(* Logix 5000 project; controller ARS14002_PLC vendor 1 type 14 code 218 rev 30.11; software revision 30.01; part 4 of 13 *)
(* tags used below, declared in another part *)
   ARGON_FROM_TK1100A : BOOL;
   ARGON_FROM_TK700 : BOOL;
   ARS14002_PLC_LEDStatus : INT;
   ARS14002_PLC_Slot1Status : INT;
   ARS14002_PLC_Slot2Status : INT;
   ARS14002_PLC_Slot3Status : INT;
   ARS14002_PLC_Slot4Status : INT;
   ARS14002_PLC_Slot5Status : INT;
   ARS14002_PLC_Status : INT;
   ARS_AUTORETURN_IGNORE_AUTO : BOOL;   // Turns furnace return autoswitch on or off
   ARS_COLLECT : BOOL;
   ARS_COLLECT_AUTO : BOOL;
   ARS_IDLE : BOOL;   // **future use
   ARS_Manual_Backfill : BOOL;   // **future use
   ARS_READY_TO_RECEIVE : BOOL;
   ARS_READY_TO_SEND : BOOL;
   ARS_RETURN : BOOL;
   ARS_RETURN_AUTO : BOOL;
   ARS_STANDBY : BOOL;
   AT2_ATOMIZE_FLOW : REAL;
   AT2_ATOMIZE_FLOW_ATOMIZE_SP : REAL;
   AT2_AtomizingStatus_OSF_OB : BOOL;
   AT2_AtomizingStatus_OSF_SB : BOOL;
   AT2_AtomizingStatus_OSR_OB : BOOL;
   AT2_AtomizingStatus_OSR_SB : BOOL;
   AT2_CHAMBER_PRESSURE : REAL;
   AT2_CHAMBER_PRESSURE_SP : REAL;
   AT2_COMM_STATUS_CONS : BOOL;
   AT2_COMM_STATUS_PROD : BOOL;
   AT2_END_ATOMIZATION : BOOL;
   AT2_HIBON_RUNNING : BOOL;
   AT2_INLET_FLOW : REAL;
   AT2_INLET_FLOW_BACKFILL_SP : REAL;
   AT2_INLET_VALVE_OPEN : BOOL;
   AT2_PLANT_ATOMIZING : BOOL;
   AT2_PLANT_BACKFILL : BOOL;
   AT2_PLANT_BACKFILL_TIMEOUT_TMR : TIMER;
   AT2_PLANT_COLLECT_AUTO : BOOL;
   AT2_PLANT_COMMLOSS : BOOL;
   AT2_PLANT_POST_ATOMIZE_TON : TIMER;
   AT2_PLANT_POST_ATOMIZING : BOOL;
   AT2_PLANT_POST_ATOMIZING_CHAMBER_SP : REAL;
   AT2_PLANT_RETURN_AUTO : BOOL;
   AT2_PRAXAIR_PRESSURE : REAL;
   AT2_PRAXAIR_PRESSURE_RETURN_SPH : REAL;
   AT2_PRAXAIR_PRESSURE_RETURN_SPL : REAL;
   AT2_START_ATOMIZATION : BOOL;
   AT2_V1_OPEN : BOOL;
   AT3_ATOMIZE_FLOW : REAL;
   AT3_ATOMIZE_FLOW_ATOMIZE_SP : REAL;
   AT3_ATOMIZE_VALVE_OPEN : BOOL;
   AT3_AtomizingStatus_OSF_OB : BOOL;
   AT3_AtomizingStatus_OSF_SB : BOOL;
   AT3_AtomizingStatus_OSR_OB : BOOL;
   AT3_AtomizingStatus_OSR_SB : BOOL;
   AT3_CHAMBER_PRESSURE : REAL;
   AT3_CHAMBER_PRESSURE_SP : REAL;
   AT3_COMM_STATUS_CONS : BOOL;
   AT3_COMM_STATUS_PROD : BOOL;
   AT3_END_ATOMIZATION : BOOL;
   AT3_HIBON_RUNNING : BOOL;
   AT3_INLET_FLOW : REAL;
   AT3_INLET_FLOW_BACKFILL_SP : REAL;
   AT3_INLET_VALVE_OPEN : BOOL;
   AT3_PLANT_ATOMIZING : BOOL;
   AT3_PLANT_BACKFILL : BOOL;
   AT3_PLANT_BACKFILL_TIMEOUT_TMR : TIMER;
   AT3_PLANT_COLLECT_AUTO : BOOL;
   AT3_PLANT_COMMLOSS : BOOL;
   AT3_PLANT_POST_ATOMIZE_TON : TIMER;
   AT3_PLANT_POST_ATOMIZING : BOOL;
   AT3_PLANT_POST_ATOMIZING_CHAMBER_SP : REAL;
   AT3_PLANT_RETURN_AUTO : BOOL;
   AT3_V1_OPEN : BOOL;
   Cold_Box_Idle : BOOL;   // **future use
   CP_PumpUp : BOOL;
   CP_PumpUp_PressurePermissive : BOOL;
   CYCLE_TIME_AT2_MIN : DINT;
   CYCLE_TIME_AT3_MIN : DINT;
   CYCLE_TIME_PILOT_MIN : DINT;
   CYCLE_TIME_REM_AT2_MIN : REAL;
   CYCLE_TIME_REM_AT3_MIN : REAL;
   CYCLE_TIME_REM_PILOT_MIN : REAL;
   ESTOP_1 : BOOL;   // Pump Skid E-Stops
   ESTOP_2 : BOOL;   // FAN/HXR E-Stops
   ESTOP_HMI : BOOL;
   ESTOP_PL : CM_DO_GENERIC;
   ESTOP_ResetReq : BOOL;
   ESTOP_TRIP : BOOL;
   EW_TEST_ATOMIZE : BOOL;
   FCV_1001 : CM_AO_VLV;
   FCV_1002 : CM_AO_VLV;
   FCV_202 : CM_AO_VLV;
   FT_904 : CM_AI_SCL;
   FVNR550_CommFlt_TON : TIMER;
   FVNR550_COMMLOSS : BOOL;
   FVNR550_L1Current_HoldingRegister : DINT;
   FVR800C_CommFlt_TON : TIMER;
   FVR800C_COMMLOSS : BOOL;
   FVR800C_L1Current_HoldingRegister : DINT;
   FVR800D_CommFlt_TON : TIMER;
   FVR800D_COMMLOSS : BOOL;
   FVR800D_L1Current_HoldingRegister : DINT;
   FVR_800C_COMMLOSS : BOOL;
   FVR_800C_EN : BOOL;
   FVR_800C_ManStartReq : BOOL;
   FVR_800C_ST : BOOL;
   FVR_800D_COMMLOSS : BOOL;
   FVR_800D_EN : BOOL;
   FVR_800D_ManStartReq : BOOL;
   FVR_800D_ST : BOOL;
   HEAT_TIMER1 : TIMER;
   HEAT_TIMER1_MIN : DINT;
   HEAT_TIMER1_MS : DINT;
   HEAT_TIMER1_SEC : DINT;
   HEAT_TIMER_AT2 : TIMER;
   HEAT_TIMER_AT2_MIN : DINT;
   HEAT_TIMER_AT2_MS : DINT;
   HEAT_TIMER_AT2_SEC : DINT;
   HEAT_TIMER_AT3 : TIMER;
   HEAT_TIMER_AT3_MIN : DINT;
   HEAT_TIMER_AT3_MS : DINT;
   HEAT_TIMER_AT3_SEC : DINT;
   HEAT_TIMER_PILOT : TIMER;
   HEAT_TIMER_PILOT_MIN : DINT;
   HEAT_TIMER_PILOT_MS : DINT;
   HEAT_TIMER_PILOT_SEC : DINT;
   MANUAL_ARS_LOCKOUT : BOOL;
   MCP_SLOT1_ERROR : BOOL;
   MCP_SLOT2_ERROR : BOOL;
   MCP_SLOT3_ERROR : BOOL;
   MCP_SLOT4_ERROR : BOOL;
   MCP_SLOT5_ERROR : BOOL;
   MODE_ATOMIZE : BOOL;
   MODE_IDLE : BOOL;
   MODE_STANDBY_IDLE : BOOL;
   MODE_STANDBY_PUMPUP : BOOL;
   OFF_TIMER_AT2 : TIMER;
   OFF_TIMER_AT3 : TIMER;
   OFF_TIMER_PILOT : TIMER;
   P_800C_Fault : BOOL;
   P_800D_Fault : BOOL;
   PDT_701_ALT_GAL : REAL;
   PIDE_800_InRange : BOOL;
   PILOT_ATOMIZE_VALVE_OPEN : BOOL;   // Halo Valve
   Pilot_AtomizingStatus_OSF_OB : BOOL;
   Pilot_AtomizingStatus_OSF_SB : BOOL;
   Pilot_AtomizingStatus_OSR_OB : BOOL;
   Pilot_AtomizingStatus_OSR_SB : BOOL;
   PILOT_COMM_STATUS : BOOL;
   PILOT_INLET_VALVE_OPEN : BOOL;   // Pressure Control Status (Backfill)
   PILOT_PLANT_ATOMIZING : BOOL;
   PILOT_PLANT_BACKFILL : BOOL;
   PILOT_PLANT_BACKFILL_TIMEOUT_TMR : TIMER;
   PILOT_PLANT_COLLECT_AUTO : BOOL;
   PILOT_PLANT_COMMLOSS : BOOL;
   PILOT_PLANT_POST_ATOMIZING_TON : TIMER;
   PILOT_PLANT_RETURN_AUTO : BOOL;
   PLC_S1_TOF : TIMER;
   PLC_S2_TOF : TIMER;
   PLC_S3_TOF : TIMER;
   PLC_S4_TOF : TIMER;
   PLC_S5_TOF : TIMER;
   PWHMI_AtomizingStatus_OSR_OB : BOOL;
   PWHMI_AtomizingStatus_OSR_SB : BOOL;
   PWHMI_AtomizingStatusVerified : BOOL;
   PWHMI_BackfillStatus : BOOL;   // PWHMI Atomizer(s) Backfilling
   PWHMI_IdleStatus : BOOL;   // **future use
   PWHMI_MeltingStatus : BOOL;   // **future use
   PWHMI_Post_Atomize_TMR : TIMER;
   PWHMI_Post_Collection_TMR : TIMER;
   PWHMI_StartAtomizing : TIMER;
   RCP_1000_COMMLOSS : BOOL;
   RCP_100_COMMLOSS : BOOL;
   RCP_600_COMMLOSS : BOOL;
   RCP_800_COMMLOSS : BOOL;
   Return_Stop_N2 : BOOL;
   Return_Stop_O2 : BOOL;
   TE_902 : CM_AI_SCL;
   TE_904 : CM_AI_SCL;
   TK_1100A_Low : BOOL;
   TK_700_Low : BOOL;
   TK_700_RETURN_SPH : REAL;
   TK_700_RETURN_SPH_SUB : REAL;
   TK_700_RETURN_SPL : REAL;
   TK_700_RETURN_SPL_PLUS : REAL;
   VFD800A_CommFlt_TON : TIMER;
   VFD800A_COMMLOSS : BOOL;
   VFD800A_DCBusVolts_HoldingRegister : DINT;
   VFD800B_CommFlt_TON : TIMER;
   VFD800B_COMMLOSS : BOOL;
   VFD800B_DCBusVolts_HoldingRegister : DINT;
   VFD_800A_COMMLOSS : BOOL;
   VFD_800A_EN : BOOL;
   VFD_800A_ManStartReq : BOOL;
   VFD_800A_ST : BOOL;
   VFD_800B_COMMLOSS : BOOL;
   VFD_800B_EN : BOOL;
   VFD_800B_ManStartReq : BOOL;
   VFD_800B_ST : BOOL;
   WATCHDOG_1000_TON1 : TIMER;
   WATCHDOG_1000_TON2 : TIMER;
   WATCHDOG_100_TON1 : TIMER;
   WATCHDOG_100_TON2 : TIMER;
   WATCHDOG_600_TON1 : TIMER;
   WATCHDOG_600_TON2 : TIMER;
   WATCHDOG_800_TON1 : TIMER;
   WATCHDOG_800_TON2 : TIMER;
   WATCHDOG_AT2_TO_ARS_TON1 : TIMER;
   WATCHDOG_AT3_TO_ARS_TON1 : TIMER;
   WATCHDOG_FROM_ARS_IN : BOOL;
   WATCHDOG_IN_100 : BOOL;
   WATCHDOG_IN_1000 : BOOL;
   WATCHDOG_IN_600 : BOOL;
   WATCHDOG_IN_800 : BOOL;
   WATCHDOG_OUT_100 : BOOL;
   WATCHDOG_OUT_1000 : BOOL;
   WATCHDOG_OUT_600 : BOOL;
   WATCHDOG_OUT_800 : BOOL;
   WATCHDOG_OUT_HMI : BOOL;
   WATCHDOG_OUT_MCP : BOOL;
   WATCHDOG_PILOT_TO_ARS_TON1 : TIMER;
   WATCHDOG_TOF : TIMER;
   WATCHDOG_TON : TIMER;
(* MainProgram, continued *)

ROUTINE _20_Safety_Misc   (* ladder *)
// Misc. Safety Functions
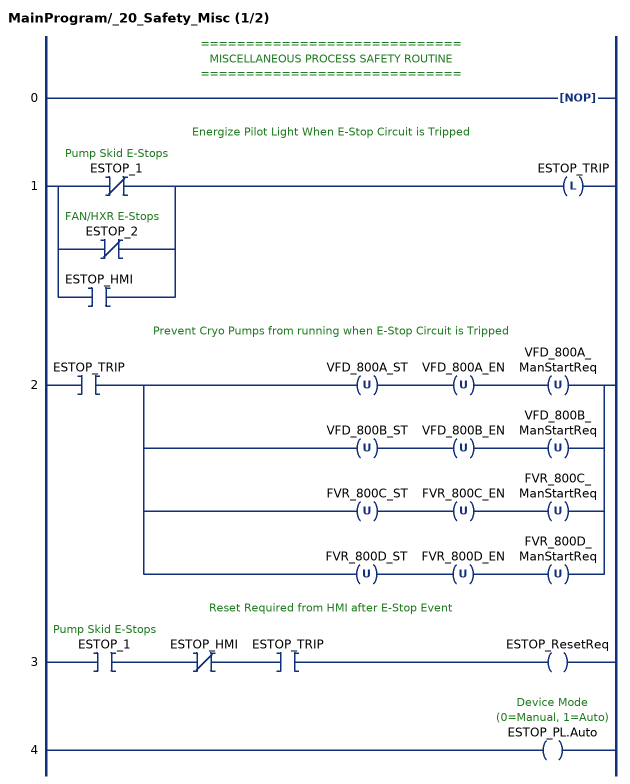
   // =============================
   // MISCELLANEOUS PROCESS SAFETY ROUTINE
   // =============================
   0: NOP();
   // Energize Pilot Light When E-Stop Circuit is Tripped
   1: [XIO(ESTOP_1) ,XIO(ESTOP_2) ,XIC(ESTOP_HMI) ]OTL(ESTOP_TRIP);
   // Prevent Cryo Pumps from running when E-Stop Circuit is Tripped
   2: XIC(ESTOP_TRIP)[OTU(VFD_800A_ST) OTU(VFD_800A_EN) OTU(VFD_800A_ManStartReq) ,OTU(VFD_800B_ST) OTU(VFD_800B_EN) OTU(VFD_800B_ManStartReq) ,OTU(FVR_800C_ST) OTU(FVR_800C_EN) OTU(FVR_800C_ManStartReq) ,OTU(FVR_800D_ST) OTU(FVR_800D_EN) OTU(FVR_800D_ManStartReq) ];
   // Reset Required from HMI after E-Stop Event
   3: XIC(ESTOP_1)XIO(ESTOP_HMI)XIC(ESTOP_TRIP)OTE(ESTOP_ResetReq);
   4: OTE(ESTOP_PL.Auto);
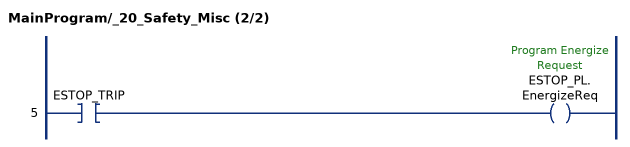
   5: XIC(ESTOP_TRIP)OTE(ESTOP_PL.EnergizeReq);
END_ROUTINE

ROUTINE _21_Watchdog   (* ladder *)
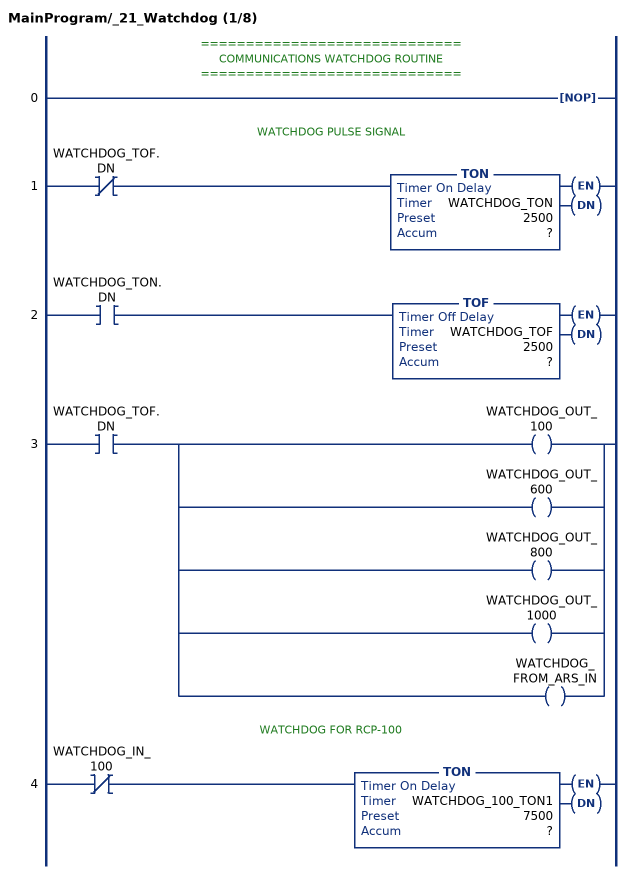
   // =============================
   // COMMUNICATIONS WATCHDOG ROUTINE
   // =============================
   0: NOP();
   // WATCHDOG PULSE SIGNAL
   1: XIO(WATCHDOG_TOF.DN)TON(WATCHDOG_TON,?,?);
   2: XIC(WATCHDOG_TON.DN)TOF(WATCHDOG_TOF,?,?);
   3: XIC(WATCHDOG_TOF.DN)[OTE(WATCHDOG_OUT_100) ,OTE(WATCHDOG_OUT_600) ,OTE(WATCHDOG_OUT_800) ,OTE(WATCHDOG_OUT_1000) ,OTE(WATCHDOG_FROM_ARS_IN) ];
   // WATCHDOG FOR RCP-100
   4: XIO(WATCHDOG_IN_100)TON(WATCHDOG_100_TON1,?,?);
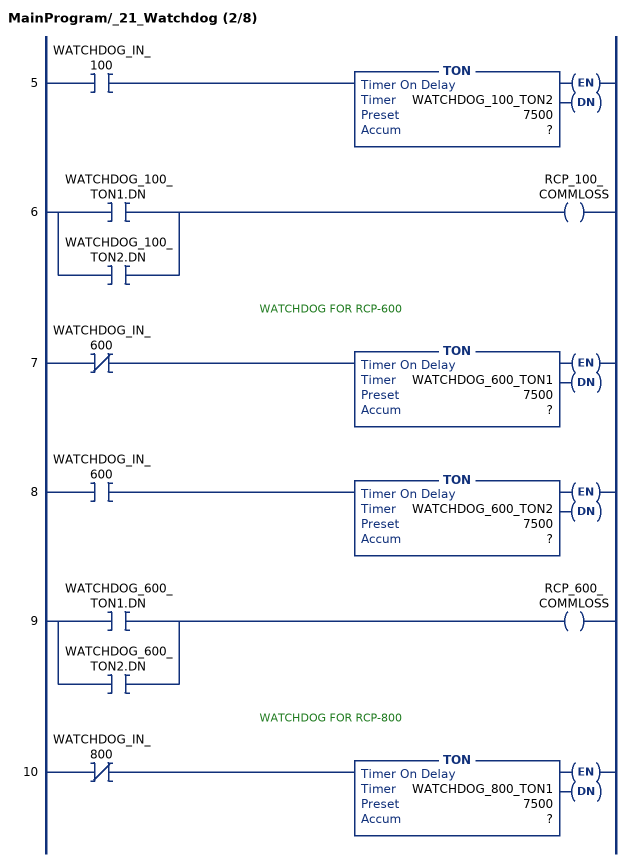
   5: XIC(WATCHDOG_IN_100)TON(WATCHDOG_100_TON2,?,?);
   6: [XIC(WATCHDOG_100_TON1.DN) ,XIC(WATCHDOG_100_TON2.DN) ]OTE(RCP_100_COMMLOSS);
   // WATCHDOG FOR RCP-600
   7: XIO(WATCHDOG_IN_600)TON(WATCHDOG_600_TON1,?,?);
   8: XIC(WATCHDOG_IN_600)TON(WATCHDOG_600_TON2,?,?);
   9: [XIC(WATCHDOG_600_TON1.DN) ,XIC(WATCHDOG_600_TON2.DN) ]OTE(RCP_600_COMMLOSS);
   // WATCHDOG FOR RCP-800
   10: XIO(WATCHDOG_IN_800)TON(WATCHDOG_800_TON1,?,?);
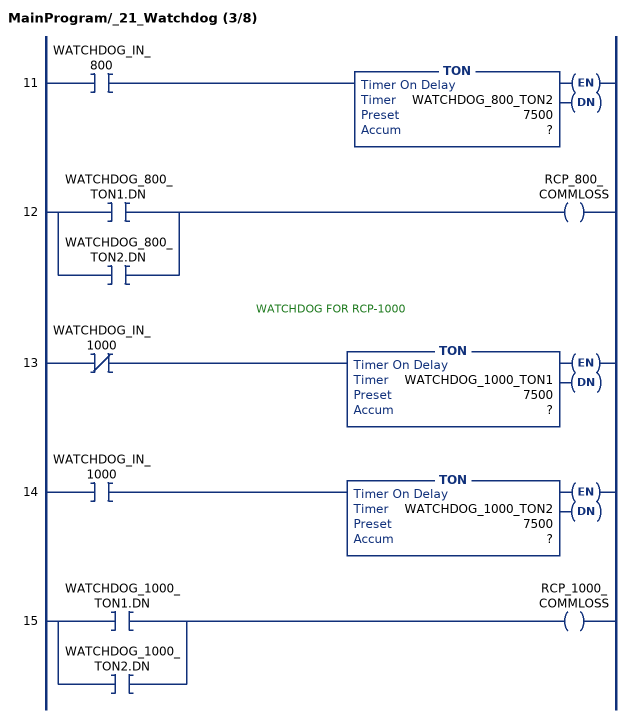
   11: XIC(WATCHDOG_IN_800)TON(WATCHDOG_800_TON2,?,?);
   12: [XIC(WATCHDOG_800_TON1.DN) ,XIC(WATCHDOG_800_TON2.DN) ]OTE(RCP_800_COMMLOSS);
   // WATCHDOG FOR RCP-1000
   13: XIO(WATCHDOG_IN_1000)TON(WATCHDOG_1000_TON1,?,?);
   14: XIC(WATCHDOG_IN_1000)TON(WATCHDOG_1000_TON2,?,?);
   15: [XIC(WATCHDOG_1000_TON1.DN) ,XIC(WATCHDOG_1000_TON2.DN) ]OTE(RCP_1000_COMMLOSS);
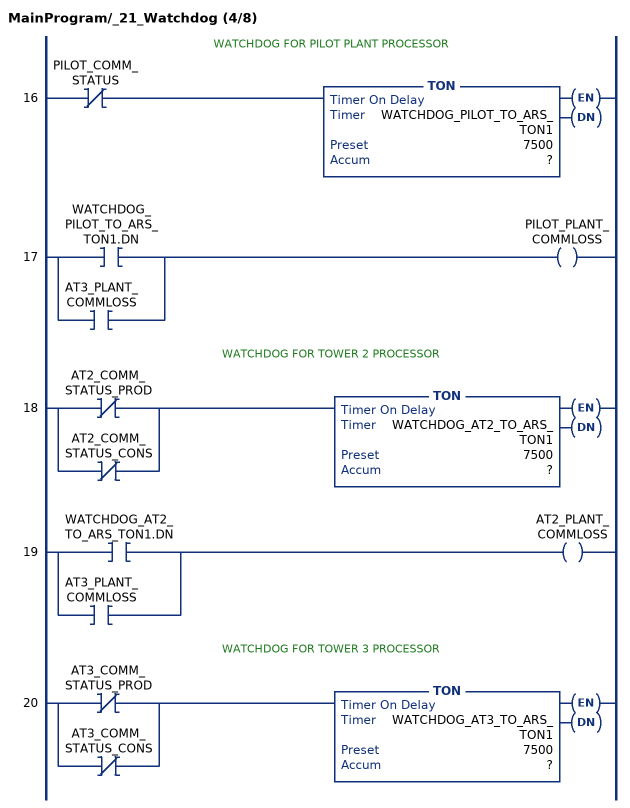
   // WATCHDOG FOR PILOT PLANT PROCESSOR
   16: XIO(PILOT_COMM_STATUS)TON(WATCHDOG_PILOT_TO_ARS_TON1,?,?);
   17: [XIC(WATCHDOG_PILOT_TO_ARS_TON1.DN) ,XIC(AT3_PLANT_COMMLOSS) ]OTE(PILOT_PLANT_COMMLOSS);
   // WATCHDOG FOR TOWER 2 PROCESSOR
   18: [XIO(AT2_COMM_STATUS_PROD) ,XIO(AT2_COMM_STATUS_CONS) ]TON(WATCHDOG_AT2_TO_ARS_TON1,?,?);
   19: [XIC(WATCHDOG_AT2_TO_ARS_TON1.DN) ,XIC(AT3_PLANT_COMMLOSS) ]OTE(AT2_PLANT_COMMLOSS);
   // WATCHDOG FOR TOWER 3 PROCESSOR
   20: [XIO(AT3_COMM_STATUS_PROD) ,XIO(AT3_COMM_STATUS_CONS) ]TON(WATCHDOG_AT3_TO_ARS_TON1,?,?);
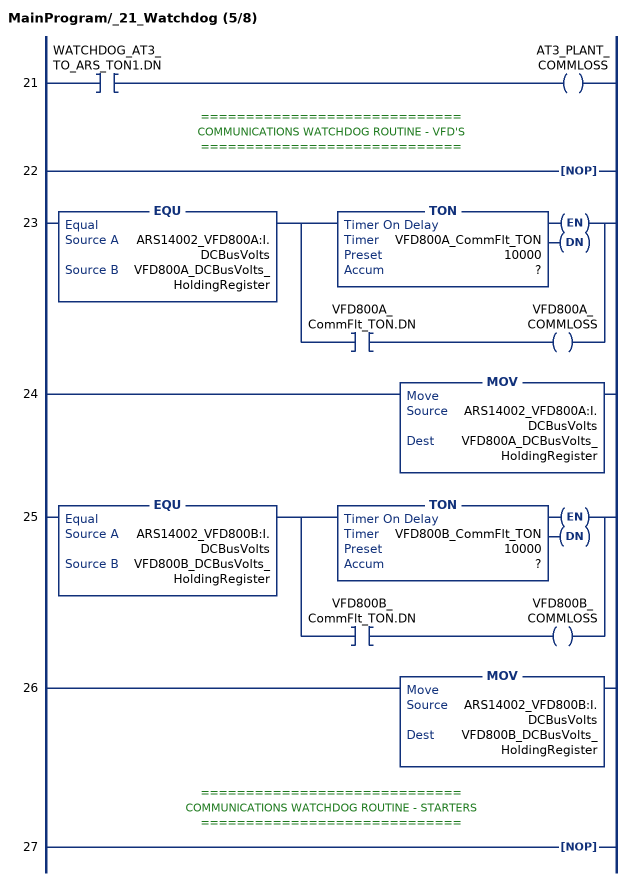
   21: XIC(WATCHDOG_AT3_TO_ARS_TON1.DN)OTE(AT3_PLANT_COMMLOSS);
   // =============================
   // COMMUNICATIONS WATCHDOG ROUTINE - VFD'S
   // =============================
   22: NOP();
   23: EQU(ARS14002_VFD800A:I.DCBusVolts,VFD800A_DCBusVolts_HoldingRegister)[TON(VFD800A_CommFlt_TON,?,?) ,XIC(VFD800A_CommFlt_TON.DN) OTE(VFD800A_COMMLOSS) ];
   24: MOV(ARS14002_VFD800A:I.DCBusVolts,VFD800A_DCBusVolts_HoldingRegister);
   25: EQU(ARS14002_VFD800B:I.DCBusVolts,VFD800B_DCBusVolts_HoldingRegister)[TON(VFD800B_CommFlt_TON,?,?) ,XIC(VFD800B_CommFlt_TON.DN) OTE(VFD800B_COMMLOSS) ];
   26: MOV(ARS14002_VFD800B:I.DCBusVolts,VFD800B_DCBusVolts_HoldingRegister);
   // =============================
   // COMMUNICATIONS WATCHDOG ROUTINE - STARTERS
   // =============================
   27: NOP();
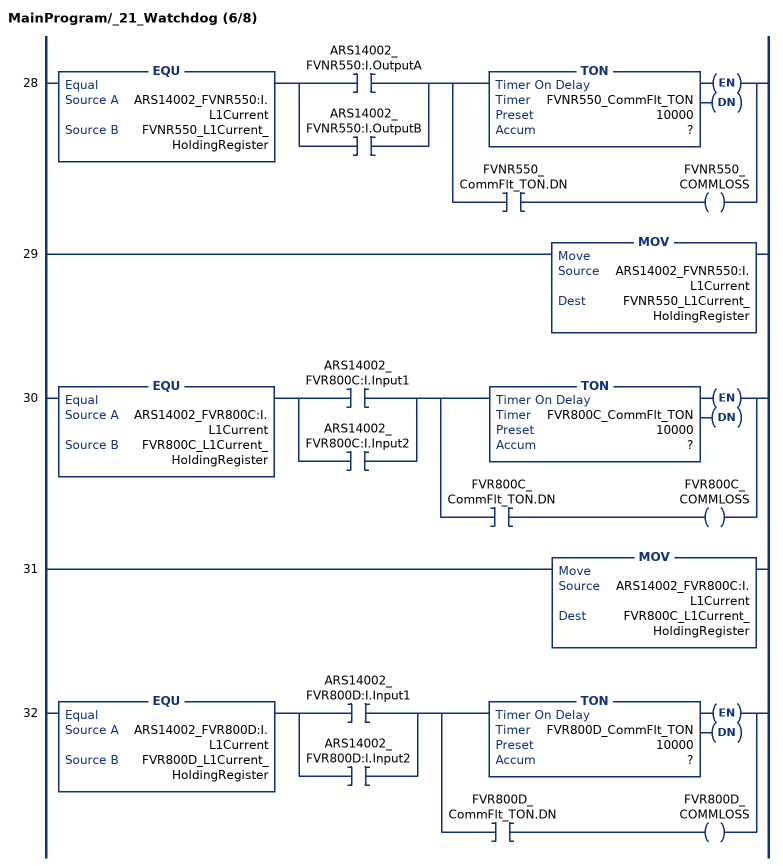
   28: EQU(ARS14002_FVNR550:I.L1Current,FVNR550_L1Current_HoldingRegister)[XIC(ARS14002_FVNR550:I.OutputA) ,XIC(ARS14002_FVNR550:I.OutputB) ][TON(FVNR550_CommFlt_TON,?,?) ,XIC(FVNR550_CommFlt_TON.DN) OTE(FVNR550_COMMLOSS) ];
   29: MOV(ARS14002_FVNR550:I.L1Current,FVNR550_L1Current_HoldingRegister);
   30: EQU(ARS14002_FVR800C:I.L1Current,FVR800C_L1Current_HoldingRegister)[XIC(ARS14002_FVR800C:I.Input1) ,XIC(ARS14002_FVR800C:I.Input2) ][TON(FVR800C_CommFlt_TON,?,?) ,XIC(FVR800C_CommFlt_TON.DN) OTE(FVR800C_COMMLOSS) ];
   31: MOV(ARS14002_FVR800C:I.L1Current,FVR800C_L1Current_HoldingRegister);
   32: EQU(ARS14002_FVR800D:I.L1Current,FVR800D_L1Current_HoldingRegister)[XIC(ARS14002_FVR800D:I.Input1) ,XIC(ARS14002_FVR800D:I.Input2) ][TON(FVR800D_CommFlt_TON,?,?) ,XIC(FVR800D_CommFlt_TON.DN) OTE(FVR800D_COMMLOSS) ];
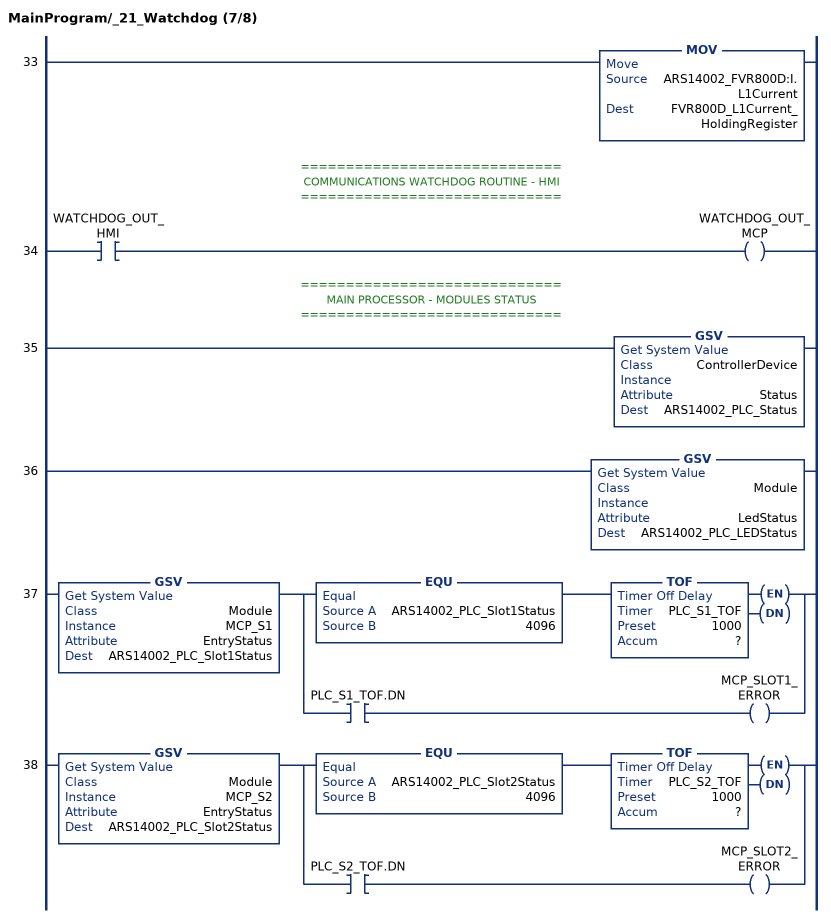
   33: MOV(ARS14002_FVR800D:I.L1Current,FVR800D_L1Current_HoldingRegister);
   // =============================
   // COMMUNICATIONS WATCHDOG ROUTINE - HMI
   // =============================
   34: XIC(WATCHDOG_OUT_HMI)OTE(WATCHDOG_OUT_MCP);
   // =============================
   // MAIN PROCESSOR - MODULES STATUS
   // =============================
   35: GSV(ControllerDevice,,Status,ARS14002_PLC_Status);
   36: GSV(Module,,LedStatus,ARS14002_PLC_LEDStatus);
   37: GSV(Module,MCP_S1,EntryStatus,ARS14002_PLC_Slot1Status)[EQU(ARS14002_PLC_Slot1Status,4096) TOF(PLC_S1_TOF,?,?) ,XIC(PLC_S1_TOF.DN) OTE(MCP_SLOT1_ERROR) ];
   38: GSV(Module,MCP_S2,EntryStatus,ARS14002_PLC_Slot2Status)[EQU(ARS14002_PLC_Slot2Status,4096) TOF(PLC_S2_TOF,?,?) ,XIC(PLC_S2_TOF.DN) OTE(MCP_SLOT2_ERROR) ];
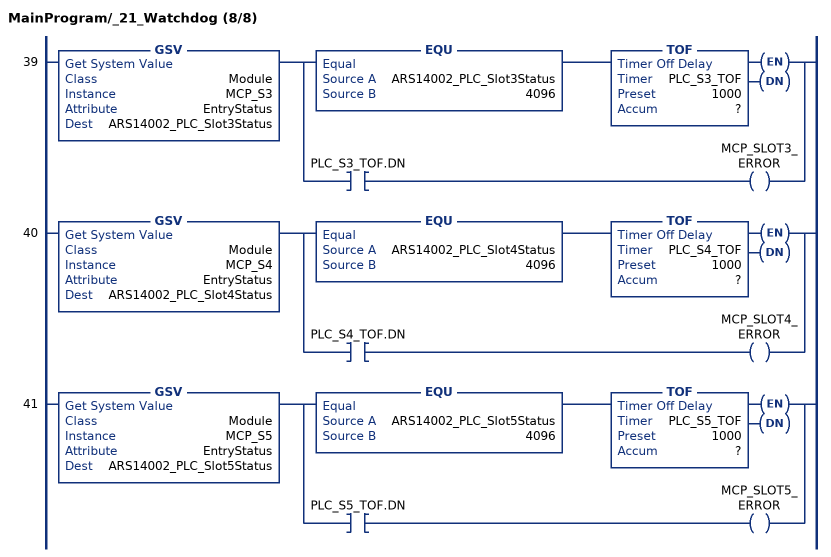
   39: GSV(Module,MCP_S3,EntryStatus,ARS14002_PLC_Slot3Status)[EQU(ARS14002_PLC_Slot3Status,4096) TOF(PLC_S3_TOF,?,?) ,XIC(PLC_S3_TOF.DN) OTE(MCP_SLOT3_ERROR) ];
   40: GSV(Module,MCP_S4,EntryStatus,ARS14002_PLC_Slot4Status)[EQU(ARS14002_PLC_Slot4Status,4096) TOF(PLC_S4_TOF,?,?) ,XIC(PLC_S4_TOF.DN) OTE(MCP_SLOT4_ERROR) ];
   41: GSV(Module,MCP_S5,EntryStatus,ARS14002_PLC_Slot5Status)[EQU(ARS14002_PLC_Slot5Status,4096) TOF(PLC_S5_TOF,?,?) ,XIC(PLC_S5_TOF.DN) OTE(MCP_SLOT5_ERROR) ];
END_ROUTINE

ROUTINE _300_Plant_Run   (* ladder *)
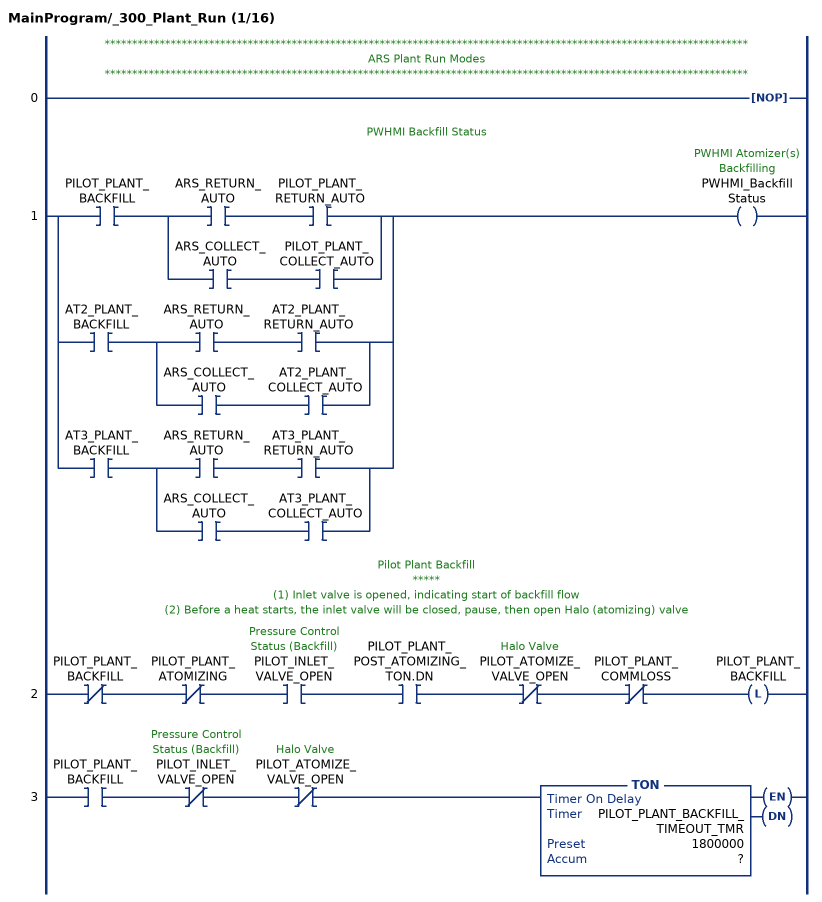
   // *********************************************************************************************************************
   // ARS Plant Run Modes
   // *********************************************************************************************************************
   0: NOP();
   // PWHMI Backfill Status
   1: [XIC(PILOT_PLANT_BACKFILL) [XIC(ARS_RETURN_AUTO) XIC(PILOT_PLANT_RETURN_AUTO) ,XIC(ARS_COLLECT_AUTO) XIC(PILOT_PLANT_COLLECT_AUTO) ] ,XIC(AT2_PLANT_BACKFILL) [XIC(ARS_RETURN_AUTO) XIC(AT2_PLANT_RETURN_AUTO) ,XIC(ARS_COLLECT_AUTO) XIC(AT2_PLANT_COLLECT_AUTO) ] ,XIC(AT3_PLANT_BACKFILL) [XIC(ARS_RETURN_AUTO) XIC(AT3_PLANT_RETURN_AUTO) ,XIC(ARS_COLLECT_AUTO) XIC(AT3_PLANT_COLLECT_AUTO) ] ]OTE(PWHMI_BackfillStatus);
   // Pilot Plant Backfill
   // *****
   // (1) Inlet valve is opened, indicating start of backfill flow
   // (2) Before a heat starts, the inlet valve will be closed, pause, then open Halo (atomizing) valve
   2: XIO(PILOT_PLANT_BACKFILL)XIO(PILOT_PLANT_ATOMIZING)XIC(PILOT_INLET_VALVE_OPEN)XIC(PILOT_PLANT_POST_ATOMIZING_TON.DN)XIO(PILOT_ATOMIZE_VALVE_OPEN)XIO(PILOT_PLANT_COMMLOSS)OTL(PILOT_PLANT_BACKFILL);
   3: XIC(PILOT_PLANT_BACKFILL)XIO(PILOT_INLET_VALVE_OPEN)XIO(PILOT_ATOMIZE_VALVE_OPEN)TON(PILOT_PLANT_BACKFILL_TIMEOUT_TMR,?,?);
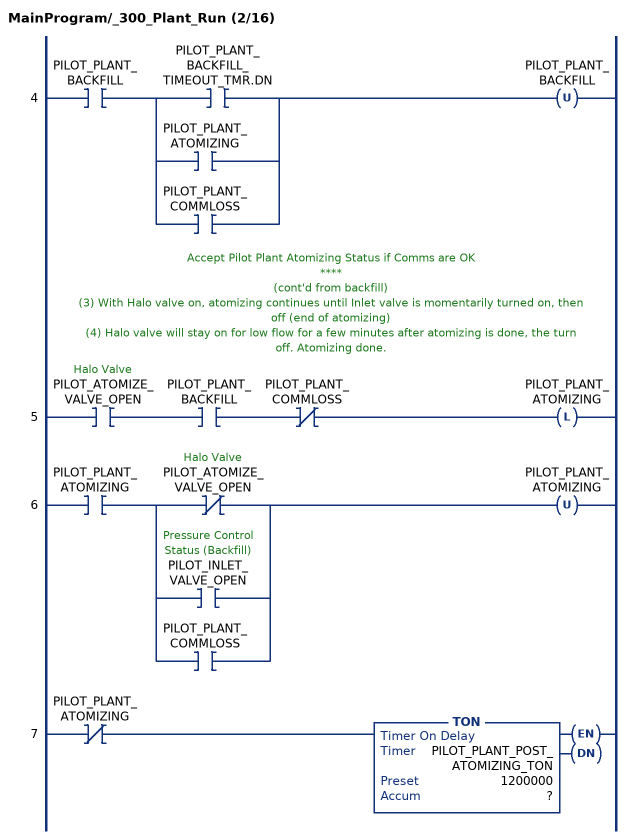
   4: XIC(PILOT_PLANT_BACKFILL)[XIC(PILOT_PLANT_BACKFILL_TIMEOUT_TMR.DN) ,XIC(PILOT_PLANT_ATOMIZING) ,XIC(PILOT_PLANT_COMMLOSS) ]OTU(PILOT_PLANT_BACKFILL);
   // Accept Pilot Plant Atomizing Status if Comms are OK
   // ****
   // (cont'd from backfill)
   // (3) With Halo valve on, atomizing continues until Inlet valve is momentarily turned on, then off (end of atomizing)
   // (4) Halo valve will stay on for low flow for a few minutes after atomizing is done, the turn off. Atomizing done.
   5: XIC(PILOT_ATOMIZE_VALVE_OPEN)XIC(PILOT_PLANT_BACKFILL)XIO(PILOT_PLANT_COMMLOSS)OTL(PILOT_PLANT_ATOMIZING);
   6: XIC(PILOT_PLANT_ATOMIZING)[XIO(PILOT_ATOMIZE_VALVE_OPEN) ,XIC(PILOT_INLET_VALVE_OPEN) ,XIC(PILOT_PLANT_COMMLOSS) ]OTU(PILOT_PLANT_ATOMIZING);
   7: XIO(PILOT_PLANT_ATOMIZING)TON(PILOT_PLANT_POST_ATOMIZING_TON,?,?);
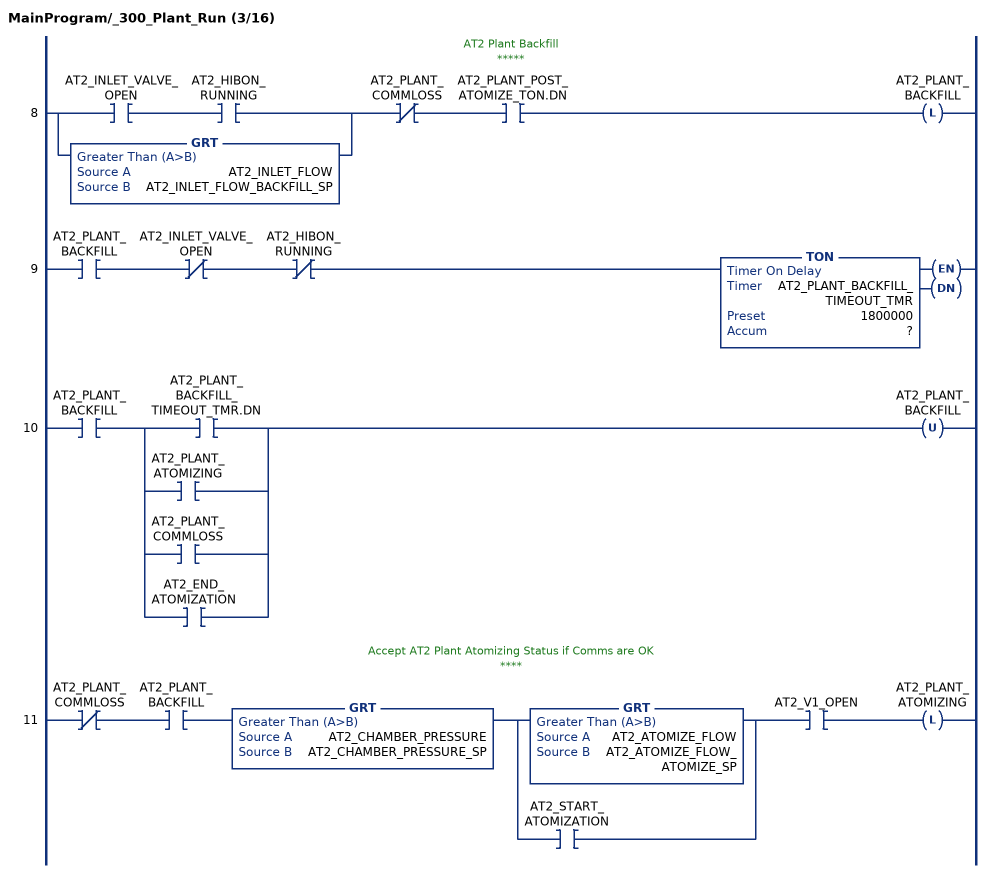
   // AT2 Plant Backfill
   // *****
   8: [XIC(AT2_INLET_VALVE_OPEN) XIC(AT2_HIBON_RUNNING) ,GRT(AT2_INLET_FLOW,AT2_INLET_FLOW_BACKFILL_SP) ]XIO(AT2_PLANT_COMMLOSS)XIC(AT2_PLANT_POST_ATOMIZE_TON.DN)OTL(AT2_PLANT_BACKFILL);
   9: XIC(AT2_PLANT_BACKFILL)XIO(AT2_INLET_VALVE_OPEN)XIO(AT2_HIBON_RUNNING)TON(AT2_PLANT_BACKFILL_TIMEOUT_TMR,?,?);
   10: XIC(AT2_PLANT_BACKFILL)[XIC(AT2_PLANT_BACKFILL_TIMEOUT_TMR.DN) ,XIC(AT2_PLANT_ATOMIZING) ,XIC(AT2_PLANT_COMMLOSS) ,XIC(AT2_END_ATOMIZATION) ]OTU(AT2_PLANT_BACKFILL);
   // Accept AT2 Plant Atomizing Status if Comms are OK
   // ****
   11: XIO(AT2_PLANT_COMMLOSS)XIC(AT2_PLANT_BACKFILL)GRT(AT2_CHAMBER_PRESSURE,AT2_CHAMBER_PRESSURE_SP)[GRT(AT2_ATOMIZE_FLOW,AT2_ATOMIZE_FLOW_ATOMIZE_SP) ,XIC(AT2_START_ATOMIZATION) ]XIC(AT2_V1_OPEN)OTL(AT2_PLANT_ATOMIZING);
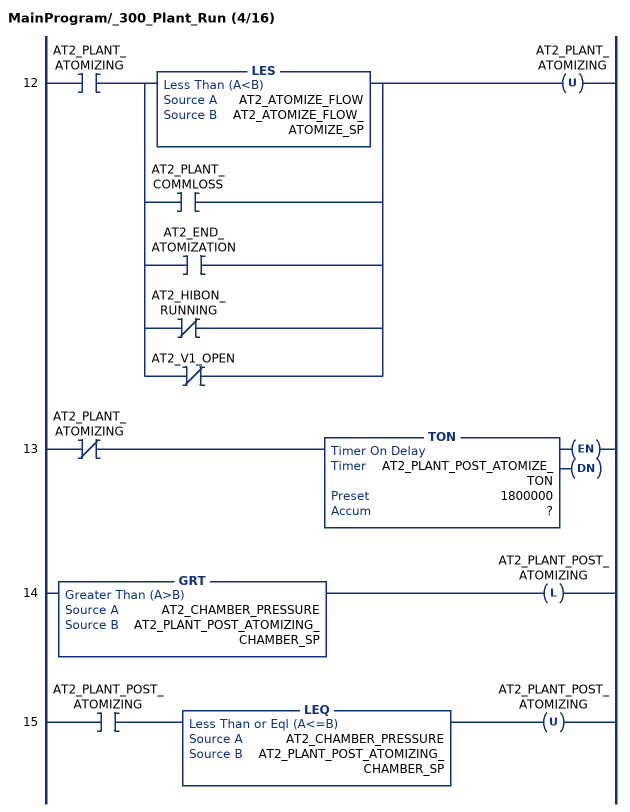
   12: XIC(AT2_PLANT_ATOMIZING)[LES(AT2_ATOMIZE_FLOW,AT2_ATOMIZE_FLOW_ATOMIZE_SP) ,XIC(AT2_PLANT_COMMLOSS) ,XIC(AT2_END_ATOMIZATION) ,XIO(AT2_HIBON_RUNNING) ,XIO(AT2_V1_OPEN) ]OTU(AT2_PLANT_ATOMIZING);
   13: XIO(AT2_PLANT_ATOMIZING)TON(AT2_PLANT_POST_ATOMIZE_TON,?,?);
   14: GRT(AT2_CHAMBER_PRESSURE,AT2_PLANT_POST_ATOMIZING_CHAMBER_SP)OTL(AT2_PLANT_POST_ATOMIZING);
   15: XIC(AT2_PLANT_POST_ATOMIZING)LEQ(AT2_CHAMBER_PRESSURE,AT2_PLANT_POST_ATOMIZING_CHAMBER_SP)OTU(AT2_PLANT_POST_ATOMIZING);
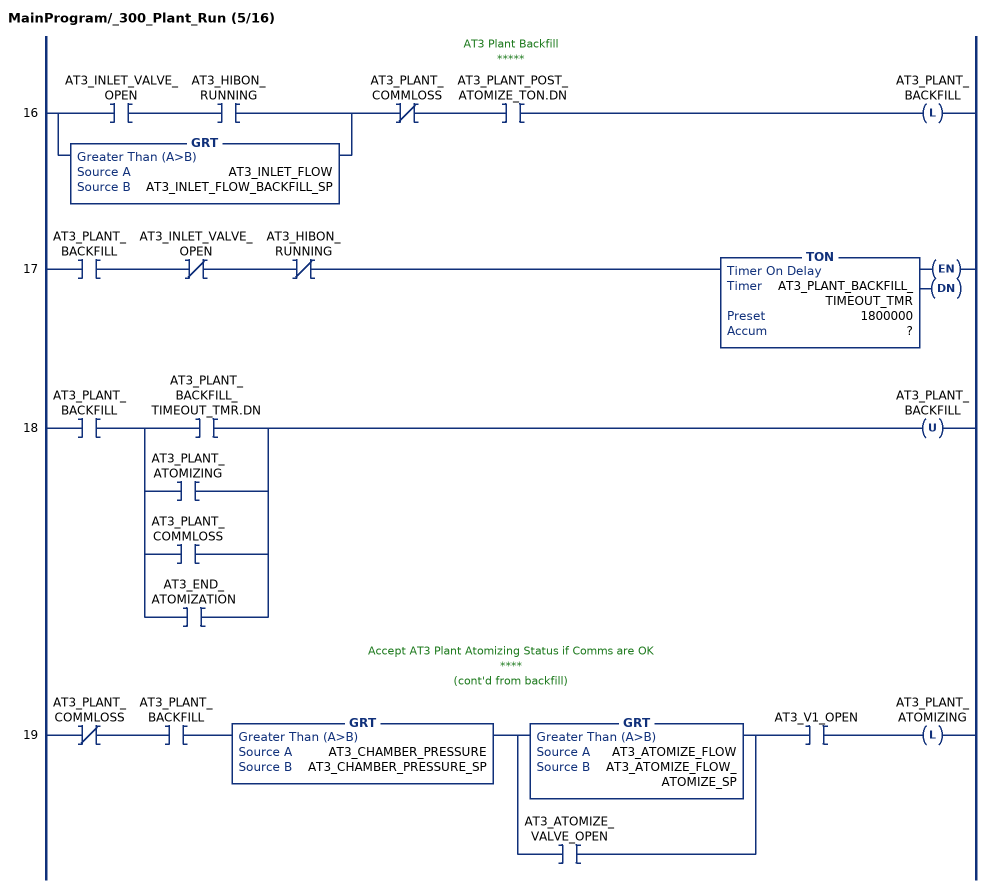
   // AT3 Plant Backfill
   // *****
   16: [XIC(AT3_INLET_VALVE_OPEN) XIC(AT3_HIBON_RUNNING) ,GRT(AT3_INLET_FLOW,AT3_INLET_FLOW_BACKFILL_SP) ]XIO(AT3_PLANT_COMMLOSS)XIC(AT3_PLANT_POST_ATOMIZE_TON.DN)OTL(AT3_PLANT_BACKFILL);
   17: XIC(AT3_PLANT_BACKFILL)XIO(AT3_INLET_VALVE_OPEN)XIO(AT3_HIBON_RUNNING)TON(AT3_PLANT_BACKFILL_TIMEOUT_TMR,?,?);
   18: XIC(AT3_PLANT_BACKFILL)[XIC(AT3_PLANT_BACKFILL_TIMEOUT_TMR.DN) ,XIC(AT3_PLANT_ATOMIZING) ,XIC(AT3_PLANT_COMMLOSS) ,XIC(AT3_END_ATOMIZATION) ]OTU(AT3_PLANT_BACKFILL);
   // Accept AT3 Plant Atomizing Status if Comms are OK
   // ****
   // (cont'd from backfill)
   19: XIO(AT3_PLANT_COMMLOSS)XIC(AT3_PLANT_BACKFILL)GRT(AT3_CHAMBER_PRESSURE,AT3_CHAMBER_PRESSURE_SP)[GRT(AT3_ATOMIZE_FLOW,AT3_ATOMIZE_FLOW_ATOMIZE_SP) ,XIC(AT3_ATOMIZE_VALVE_OPEN) ]XIC(AT3_V1_OPEN)OTL(AT3_PLANT_ATOMIZING);
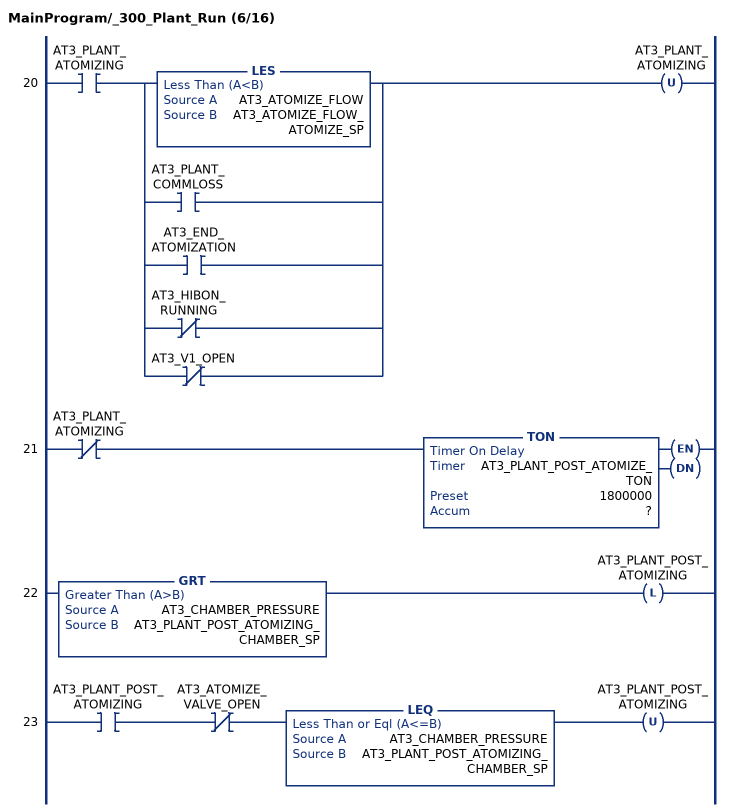
   20: XIC(AT3_PLANT_ATOMIZING)[LES(AT3_ATOMIZE_FLOW,AT3_ATOMIZE_FLOW_ATOMIZE_SP) ,XIC(AT3_PLANT_COMMLOSS) ,XIC(AT3_END_ATOMIZATION) ,XIO(AT3_HIBON_RUNNING) ,XIO(AT3_V1_OPEN) ]OTU(AT3_PLANT_ATOMIZING);
   21: XIO(AT3_PLANT_ATOMIZING)TON(AT3_PLANT_POST_ATOMIZE_TON,?,?);
   22: GRT(AT3_CHAMBER_PRESSURE,AT3_PLANT_POST_ATOMIZING_CHAMBER_SP)OTL(AT3_PLANT_POST_ATOMIZING);
   23: XIC(AT3_PLANT_POST_ATOMIZING)XIO(AT3_ATOMIZE_VALVE_OPEN)LEQ(AT3_CHAMBER_PRESSURE,AT3_PLANT_POST_ATOMIZING_CHAMBER_SP)OTU(AT3_PLANT_POST_ATOMIZING);
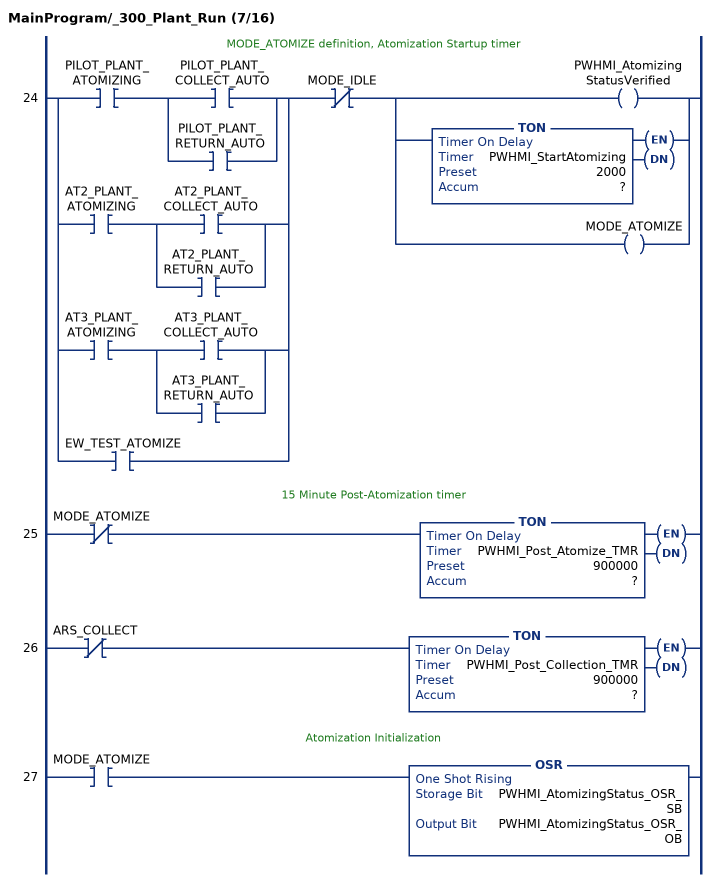
   // MODE_ATOMIZE definition, Atomization Startup timer
   24: [XIC(PILOT_PLANT_ATOMIZING) [XIC(PILOT_PLANT_COLLECT_AUTO) ,XIC(PILOT_PLANT_RETURN_AUTO) ] ,XIC(AT2_PLANT_ATOMIZING) [XIC(AT2_PLANT_COLLECT_AUTO) ,XIC(AT2_PLANT_RETURN_AUTO) ] ,[XIC(AT3_PLANT_ATOMIZING) [XIC(AT3_PLANT_COLLECT_AUTO) ,XIC(AT3_PLANT_RETURN_AUTO) ] ,XIC(EW_TEST_ATOMIZE) ] ]XIO(MODE_IDLE)[OTE(PWHMI_AtomizingStatusVerified) ,TON(PWHMI_StartAtomizing,?,?) ,OTE(MODE_ATOMIZE) ];
   // 15 Minute Post-Atomization timer
   25: XIO(MODE_ATOMIZE)TON(PWHMI_Post_Atomize_TMR,?,?);
   26: XIO(ARS_COLLECT)TON(PWHMI_Post_Collection_TMR,?,?);
   // Atomization Initialization
   27: XIC(MODE_ATOMIZE)OSR(PWHMI_AtomizingStatus_OSR_SB,PWHMI_AtomizingStatus_OSR_OB);
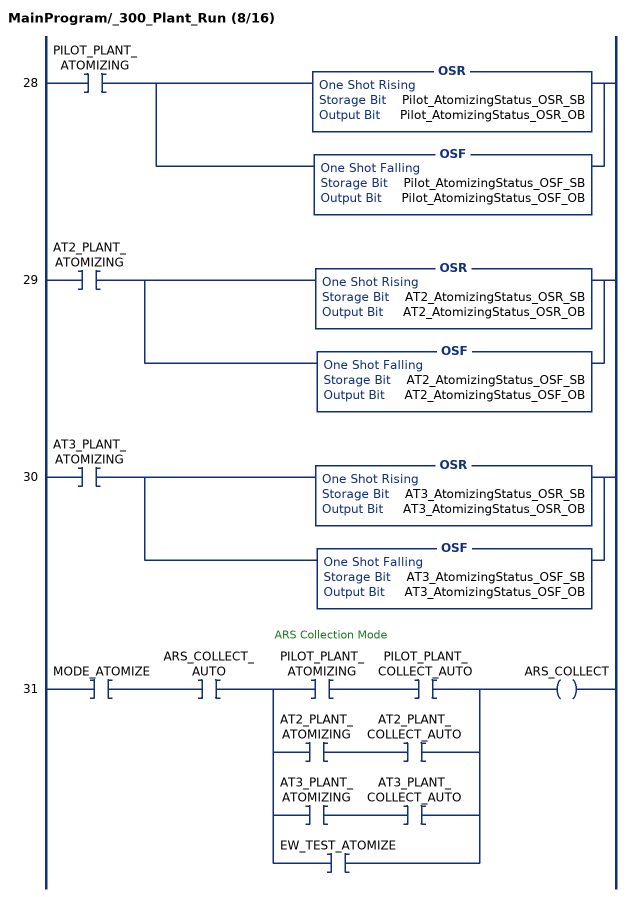
   28: XIC(PILOT_PLANT_ATOMIZING)[OSR(Pilot_AtomizingStatus_OSR_SB,Pilot_AtomizingStatus_OSR_OB) ,OSF(Pilot_AtomizingStatus_OSF_SB,Pilot_AtomizingStatus_OSF_OB) ];
   29: XIC(AT2_PLANT_ATOMIZING)[OSR(AT2_AtomizingStatus_OSR_SB,AT2_AtomizingStatus_OSR_OB) ,OSF(AT2_AtomizingStatus_OSF_SB,AT2_AtomizingStatus_OSF_OB) ];
   30: XIC(AT3_PLANT_ATOMIZING)[OSR(AT3_AtomizingStatus_OSR_SB,AT3_AtomizingStatus_OSR_OB) ,OSF(AT3_AtomizingStatus_OSF_SB,AT3_AtomizingStatus_OSF_OB) ];
   // ARS Collection Mode
   31: XIC(MODE_ATOMIZE)XIC(ARS_COLLECT_AUTO)[XIC(PILOT_PLANT_ATOMIZING) XIC(PILOT_PLANT_COLLECT_AUTO) ,XIC(AT2_PLANT_ATOMIZING) XIC(AT2_PLANT_COLLECT_AUTO) ,[XIC(AT3_PLANT_ATOMIZING) XIC(AT3_PLANT_COLLECT_AUTO) ,XIC(EW_TEST_ATOMIZE) ] ]OTE(ARS_COLLECT);
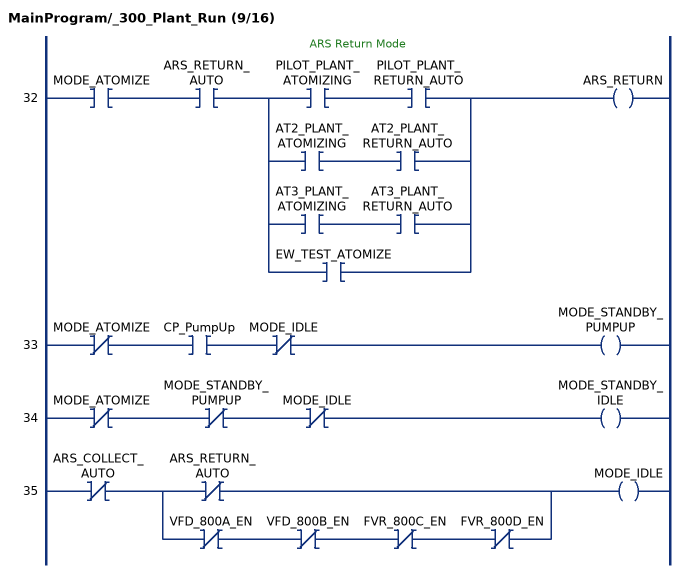
   // ARS Return Mode
   32: XIC(MODE_ATOMIZE)XIC(ARS_RETURN_AUTO)[XIC(PILOT_PLANT_ATOMIZING) XIC(PILOT_PLANT_RETURN_AUTO) ,XIC(AT2_PLANT_ATOMIZING) XIC(AT2_PLANT_RETURN_AUTO) ,[XIC(AT3_PLANT_ATOMIZING) XIC(AT3_PLANT_RETURN_AUTO) ,XIC(EW_TEST_ATOMIZE) ] ]OTE(ARS_RETURN);
   33: XIO(MODE_ATOMIZE)XIC(CP_PumpUp)XIO(MODE_IDLE)OTE(MODE_STANDBY_PUMPUP);
   34: XIO(MODE_ATOMIZE)XIO(MODE_STANDBY_PUMPUP)XIO(MODE_IDLE)OTE(MODE_STANDBY_IDLE);
   35: XIO(ARS_COLLECT_AUTO)[XIO(ARS_RETURN_AUTO) ,XIO(VFD_800A_EN) XIO(VFD_800B_EN) XIO(FVR_800C_EN) XIO(FVR_800D_EN) ]OTE(MODE_IDLE);
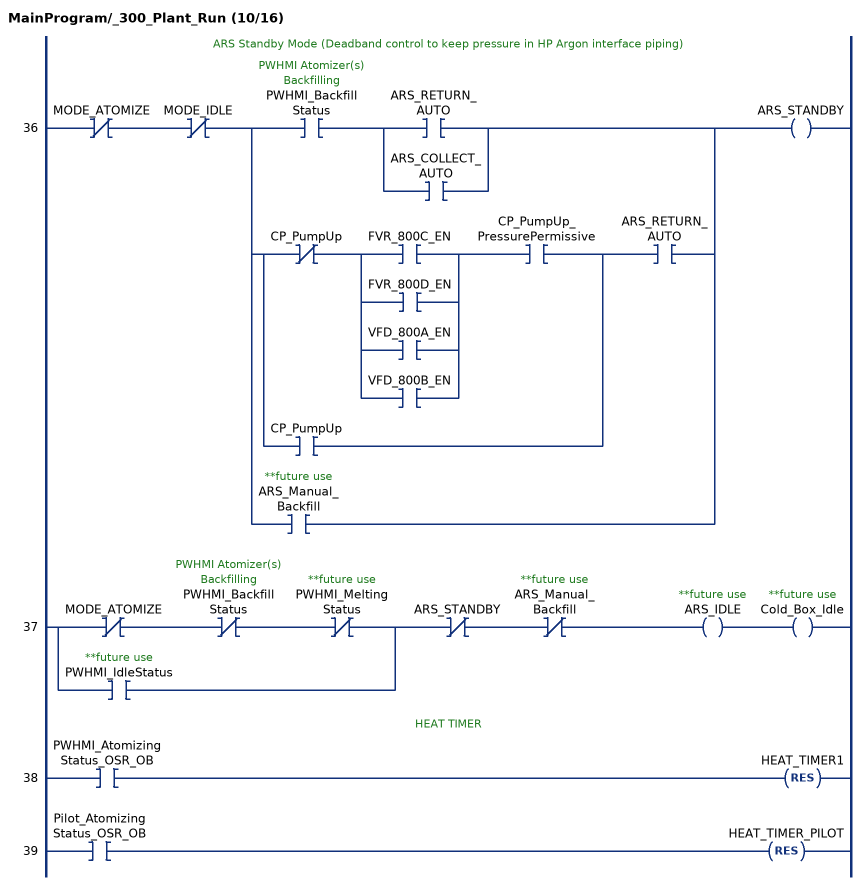
   // ARS Standby Mode (Deadband control to keep pressure in HP Argon interface piping)
   36: XIO(MODE_ATOMIZE)XIO(MODE_IDLE)[[XIC(PWHMI_BackfillStatus) [XIC(ARS_RETURN_AUTO) ,XIC(ARS_COLLECT_AUTO) ] ,[XIO(CP_PumpUp) [XIC(FVR_800C_EN) ,XIC(FVR_800D_EN) ,XIC(VFD_800A_EN) ,XIC(VFD_800B_EN) ] XIC(CP_PumpUp_PressurePermissive) ,XIC(CP_PumpUp) ] XIC(ARS_RETURN_AUTO) ] ,XIC(ARS_Manual_Backfill) ]OTE(ARS_STANDBY);
   37: [XIO(MODE_ATOMIZE) XIO(PWHMI_BackfillStatus) XIO(PWHMI_MeltingStatus) ,XIC(PWHMI_IdleStatus) ]XIO(ARS_STANDBY)XIO(ARS_Manual_Backfill)OTE(ARS_IDLE)OTE(Cold_Box_Idle);
   // HEAT TIMER
   38: XIC(PWHMI_AtomizingStatus_OSR_OB)RES(HEAT_TIMER1);
   39: XIC(Pilot_AtomizingStatus_OSR_OB)RES(HEAT_TIMER_PILOT);
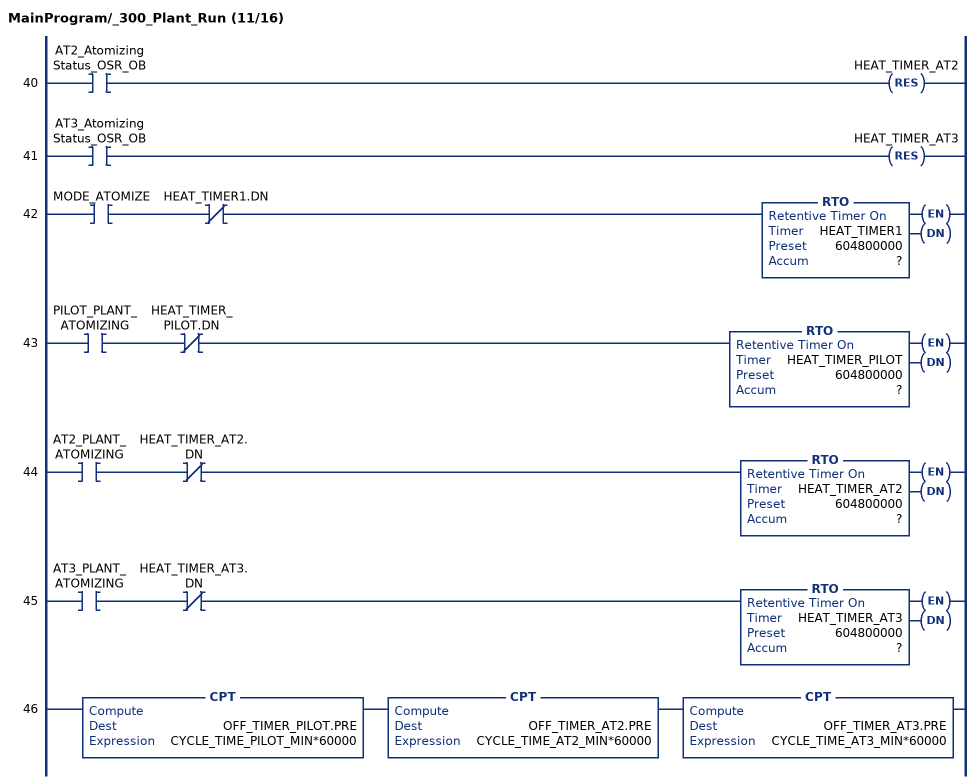
   40: XIC(AT2_AtomizingStatus_OSR_OB)RES(HEAT_TIMER_AT2);
   41: XIC(AT3_AtomizingStatus_OSR_OB)RES(HEAT_TIMER_AT3);
   42: XIC(MODE_ATOMIZE)XIO(HEAT_TIMER1.DN)RTO(HEAT_TIMER1,?,?);
   43: XIC(PILOT_PLANT_ATOMIZING)XIO(HEAT_TIMER_PILOT.DN)RTO(HEAT_TIMER_PILOT,?,?);
   44: XIC(AT2_PLANT_ATOMIZING)XIO(HEAT_TIMER_AT2.DN)RTO(HEAT_TIMER_AT2,?,?);
   45: XIC(AT3_PLANT_ATOMIZING)XIO(HEAT_TIMER_AT3.DN)RTO(HEAT_TIMER_AT3,?,?);
   46: CPT(OFF_TIMER_PILOT.PRE,CYCLE_TIME_PILOT_MIN*60000)CPT(OFF_TIMER_AT2.PRE,CYCLE_TIME_AT2_MIN*60000)CPT(OFF_TIMER_AT3.PRE,CYCLE_TIME_AT3_MIN*60000);
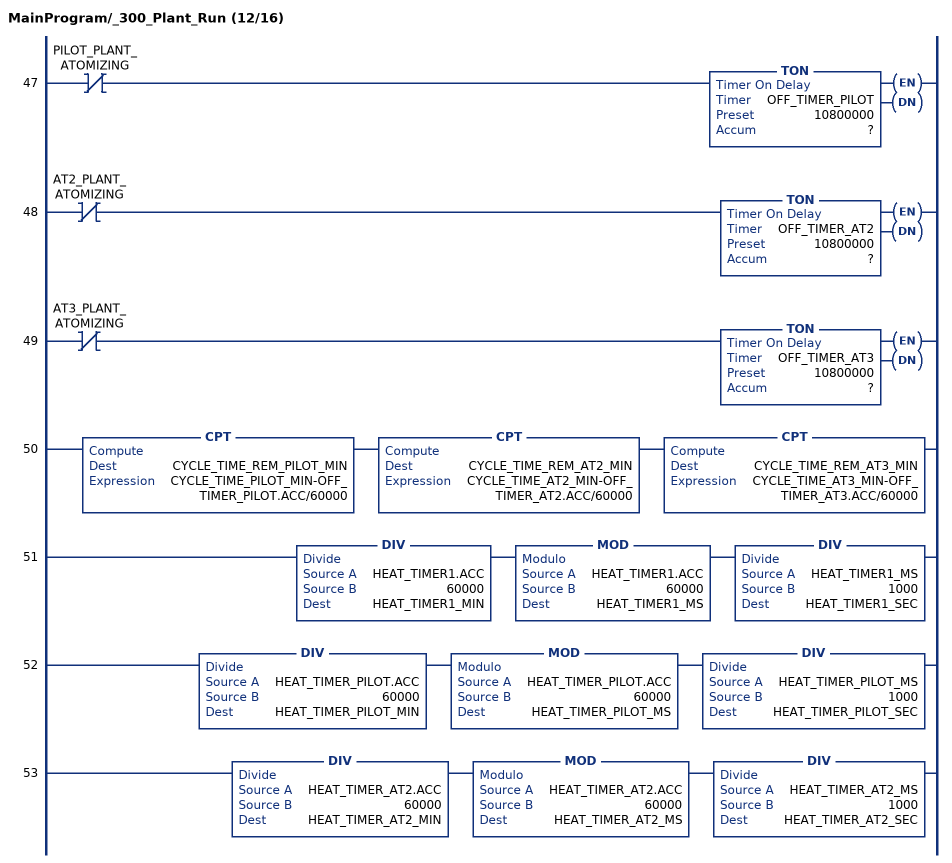
   47: XIO(PILOT_PLANT_ATOMIZING)TON(OFF_TIMER_PILOT,?,?);
   48: XIO(AT2_PLANT_ATOMIZING)TON(OFF_TIMER_AT2,?,?);
   49: XIO(AT3_PLANT_ATOMIZING)TON(OFF_TIMER_AT3,?,?);
   50: CPT(CYCLE_TIME_REM_PILOT_MIN,CYCLE_TIME_PILOT_MIN-OFF_TIMER_PILOT.ACC/60000)CPT(CYCLE_TIME_REM_AT2_MIN,CYCLE_TIME_AT2_MIN-OFF_TIMER_AT2.ACC/60000)CPT(CYCLE_TIME_REM_AT3_MIN,CYCLE_TIME_AT3_MIN-OFF_TIMER_AT3.ACC/60000);
   51: DIV(HEAT_TIMER1.ACC,60000,HEAT_TIMER1_MIN)MOD(HEAT_TIMER1.ACC,60000,HEAT_TIMER1_MS)DIV(HEAT_TIMER1_MS,1000,HEAT_TIMER1_SEC);
   52: DIV(HEAT_TIMER_PILOT.ACC,60000,HEAT_TIMER_PILOT_MIN)MOD(HEAT_TIMER_PILOT.ACC,60000,HEAT_TIMER_PILOT_MS)DIV(HEAT_TIMER_PILOT_MS,1000,HEAT_TIMER_PILOT_SEC);
   53: DIV(HEAT_TIMER_AT2.ACC,60000,HEAT_TIMER_AT2_MIN)MOD(HEAT_TIMER_AT2.ACC,60000,HEAT_TIMER_AT2_MS)DIV(HEAT_TIMER_AT2_MS,1000,HEAT_TIMER_AT2_SEC);
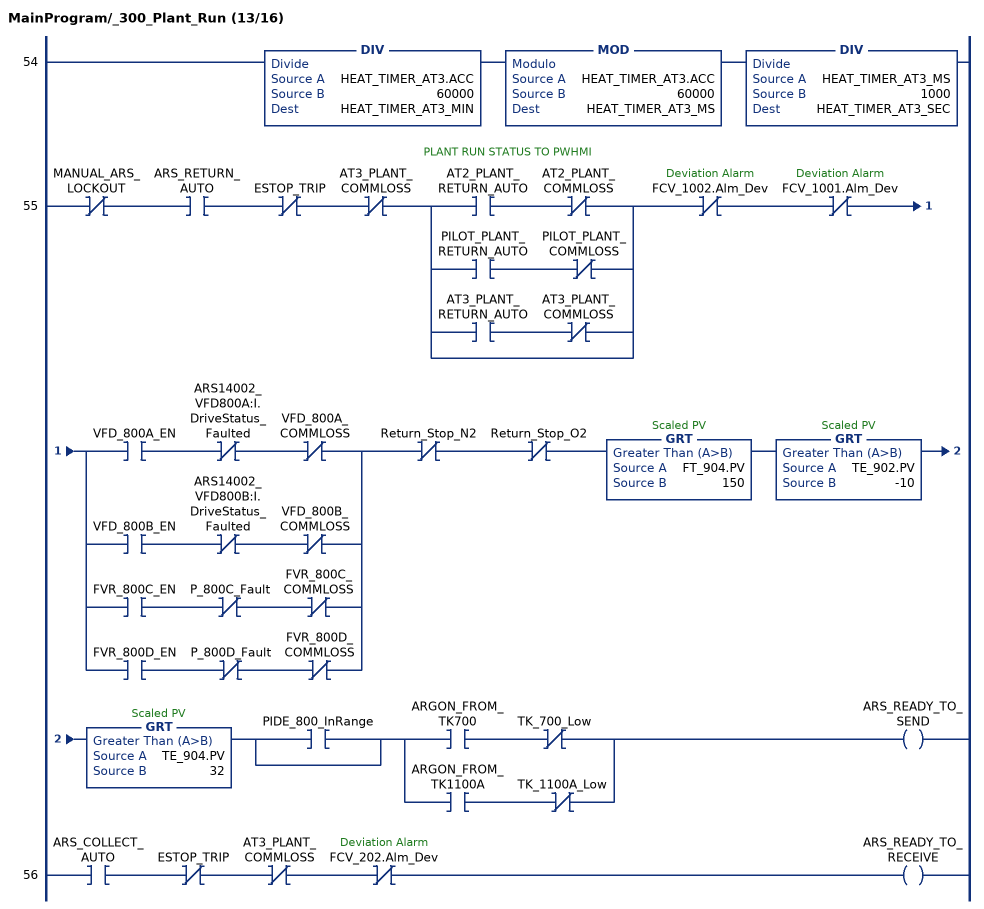
   54: DIV(HEAT_TIMER_AT3.ACC,60000,HEAT_TIMER_AT3_MIN)MOD(HEAT_TIMER_AT3.ACC,60000,HEAT_TIMER_AT3_MS)DIV(HEAT_TIMER_AT3_MS,1000,HEAT_TIMER_AT3_SEC);
   // PLANT RUN STATUS TO PWHMI
   55: XIO(MANUAL_ARS_LOCKOUT)XIC(ARS_RETURN_AUTO)XIO(ESTOP_TRIP)XIO(AT3_PLANT_COMMLOSS)[XIC(AT2_PLANT_RETURN_AUTO) XIO(AT2_PLANT_COMMLOSS) ,XIC(PILOT_PLANT_RETURN_AUTO) XIO(PILOT_PLANT_COMMLOSS) ,XIC(AT3_PLANT_RETURN_AUTO) XIO(AT3_PLANT_COMMLOSS) ,]XIO(FCV_1002.Alm_Dev)XIO(FCV_1001.Alm_Dev)[XIC(VFD_800A_EN) XIO(ARS14002_VFD800A:I.DriveStatus_Faulted) XIO(VFD_800A_COMMLOSS) ,XIC(VFD_800B_EN) XIO(ARS14002_VFD800B:I.DriveStatus_Faulted) XIO(VFD_800B_COMMLOSS) ,XIC(FVR_800C_EN) XIO(P_800C_Fault) XIO(FVR_800C_COMMLOSS) ,XIC(FVR_800D_EN) XIO(P_800D_Fault) XIO(FVR_800D_COMMLOSS) ]XIO(Return_Stop_N2)XIO(Return_Stop_O2)GRT(FT_904.PV,150)GRT(TE_902.PV,-10)GRT(TE_904.PV,32)[XIC(PIDE_800_InRange) ,][XIC(ARGON_FROM_TK700) XIO(TK_700_Low) ,XIC(ARGON_FROM_TK1100A) XIO(TK_1100A_Low) ]OTE(ARS_READY_TO_SEND);
   56: XIC(ARS_COLLECT_AUTO)XIO(ESTOP_TRIP)XIO(AT3_PLANT_COMMLOSS)XIO(FCV_202.Alm_Dev)OTE(ARS_READY_TO_RECEIVE);
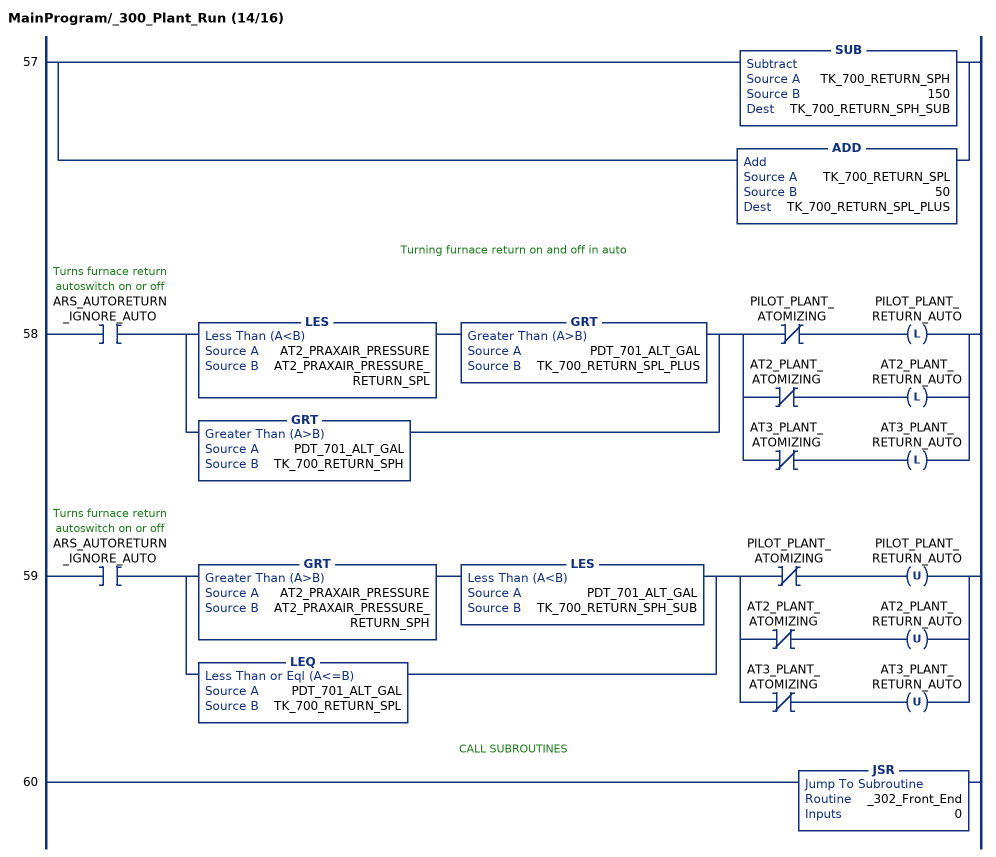
   57: [SUB(TK_700_RETURN_SPH,150,TK_700_RETURN_SPH_SUB) ,ADD(TK_700_RETURN_SPL,50,TK_700_RETURN_SPL_PLUS) ];
   // Turning furnace return on and off in auto
   58: XIC(ARS_AUTORETURN_IGNORE_AUTO)[LES(AT2_PRAXAIR_PRESSURE,AT2_PRAXAIR_PRESSURE_RETURN_SPL) GRT(PDT_701_ALT_GAL,TK_700_RETURN_SPL_PLUS) ,GRT(PDT_701_ALT_GAL,TK_700_RETURN_SPH) ][XIO(PILOT_PLANT_ATOMIZING) OTL(PILOT_PLANT_RETURN_AUTO) ,XIO(AT2_PLANT_ATOMIZING) OTL(AT2_PLANT_RETURN_AUTO) ,XIO(AT3_PLANT_ATOMIZING) OTL(AT3_PLANT_RETURN_AUTO) ];
   59: XIC(ARS_AUTORETURN_IGNORE_AUTO)[GRT(AT2_PRAXAIR_PRESSURE,AT2_PRAXAIR_PRESSURE_RETURN_SPH) LES(PDT_701_ALT_GAL,TK_700_RETURN_SPH_SUB) ,LEQ(PDT_701_ALT_GAL,TK_700_RETURN_SPL) ][XIO(PILOT_PLANT_ATOMIZING) OTU(PILOT_PLANT_RETURN_AUTO) ,XIO(AT2_PLANT_ATOMIZING) OTU(AT2_PLANT_RETURN_AUTO) ,XIO(AT3_PLANT_ATOMIZING) OTU(AT3_PLANT_RETURN_AUTO) ];
   // CALL SUBROUTINES
   60: JSR(_302_Front_End,0);
